FUNCTION_BLOCK Area_CAT (* Composite Function Block Type *)
  (* Standard: 61499-2 *)
  (* Version 0.0, 7/23/2025, Evans_A, Schneider Electric, template *)
  PACKAGE Main;
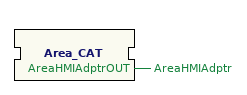
  PLUGS
    AreaHMIAdptrOUT : AreaHMIAdptr;
  END_PLUGS
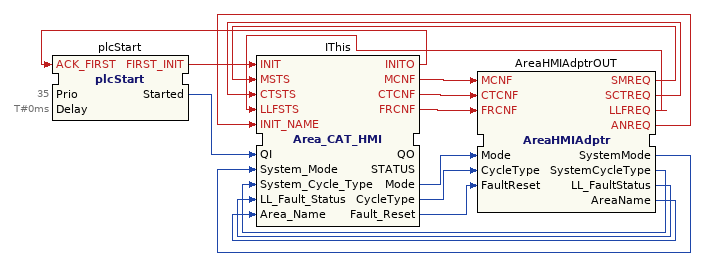
  FBS
    IThis : Area_CAT_HMI;
    plcStart : plcStart(Prio := 35, Delay := T#0ms);
  END_FBS
  EVENT_CONNECTIONS
    plcStart.FIRST_INIT TO IThis.INIT;
    AreaHMIAdptrOUT.SMREQ TO IThis.MSTS;
    AreaHMIAdptrOUT.SCTREQ TO IThis.CTSTS;
    AreaHMIAdptrOUT.LLFREQ TO IThis.LLFSTS;
    AreaHMIAdptrOUT.ANREQ TO IThis.INIT_NAME;
    IThis.INITO TO plcStart.ACK_FIRST;
    IThis.MCNF TO AreaHMIAdptrOUT.MCNF;
    IThis.CTCNF TO AreaHMIAdptrOUT.CTCNF;
    IThis.FRCNF TO AreaHMIAdptrOUT.FRCNF;
  END_CONNECTIONS
  DATA_CONNECTIONS
    plcStart.Started TO IThis.QI;
    AreaHMIAdptrOUT.SystemMode TO IThis.System_Mode;
    AreaHMIAdptrOUT.SystemCycleType TO IThis.System_Cycle_Type;
    AreaHMIAdptrOUT.LL_FaultStatus TO IThis.LL_Fault_Status;
    AreaHMIAdptrOUT.AreaName TO IThis.Area_Name;
    IThis.Mode TO AreaHMIAdptrOUT.Mode;
    IThis.CycleType TO AreaHMIAdptrOUT.CycleType;
    IThis.Fault_Reset TO AreaHMIAdptrOUT.FaultReset;
  END_CONNECTIONS
END_FUNCTION_BLOCK
